Staubli VAL3: chinese.dtx

public string No = "No"
public string Yes = "Yes "
